Fanuc KAREL source: kb00134.KL

-- PROVISIONAL review KL for V1013-1; original PC SHA256 8fc7f8dc7265d9dc075e6c679cd1b9de5e0780dc886e5bd2ae66a875cc0daaf5
-- Incomplete behavior may be omitted. Consult companion uncertainty JSON. Do not deploy.
PROGRAM KB00134
%NOLOCKGROUP
BEGIN
  -- UNRESOLVED_PC offsets 5-12; opcodes 9D,23
  -- UNRESOLVED_PC offsets 17-26; opcodes 3F,75
  -- UNRESOLVED_PC offsets 31-38; opcodes 9D,23
  -- UNRESOLVED_PC offsets 43-50; opcodes 9D,23
  -- UNRESOLVED_PC offsets 55-85; opcodes 27,22,22,2A,22,22,31
  -- UNRESOLVED_PC offsets 90-94; opcodes 7F
END KB00134
